FUNCTION_BLOCK MECHC_VIEWL (* Linear Mechanism View with Clamping & Local Data Publish/Subscribe *)
  (* Standard: 61499-1; Classification: View *)
  (* Version 0.2, 2004-10-06, JHC, Rockwell Automation, Added CNV input. *)
  (* Version 0.1, 2004-09-27, JHC, Rockwell Automation, Changed order of REND vars for consitency with MECH_VIEWL.. *)
  (* Version 0.0, 2002-05-21, JHC, Rockwell Automation, Copied/Modified from MECH_VIEWL. *)
  (* Compiler header: package fb.rt.mva; import fb.rt.net.*; *)
  (* Compiler classdef: public class MECHC_VIEWL extends FBMVCD *)
  (* Compiler Java Sun JDK 1.4.2 *)
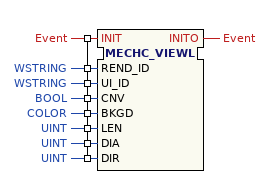
  EVENT_INPUT
    INIT WITH REND_ID, UI_ID, BKGD, LEN, DIA, DIR, CNV; (* Initialize *)
  END_EVENT
  EVENT_OUTPUT
    INITO; (* Initialized *)
  END_EVENT
  VAR_INPUT
    REND_ID : WSTRING; (* Rendering Data Channel from Model *)
    UI_ID : WSTRING; (* User Input Channel to Model *)
    CNV : BOOL; (* 0=Paint workpiece with clamp,1=Paint as conveyor with gate at end. *)
    BKGD : COLOR := blue; (* Background Color *)
    LEN : UINT; (* Length in Diameters *)
    DIA : UINT; (* Diameter *)
    DIR : UINT; (* Orientation:0=L/R,1=T/B,2=R/L,3=B/T *)
  END_VAR
  FBS
    REND : SUBL_4;
    VIEW : MECHC_VIEW;
    UI : PUBL_1;
  END_FBS
  EVENT_CONNECTIONS
    INIT TO REND.INIT;
    REND.INITO TO VIEW.INIT;
    VIEW.INITO TO UI.INIT;
    UI.INITO TO INITO;
    REND.IND TO VIEW.REQ;
    VIEW.IND TO UI.REQ;
  END_CONNECTIONS
  DATA_CONNECTIONS
    REND.RD_1 TO VIEW.POS;
    VIEW.FAULT TO UI.SD_1;
    REND_ID TO REND.ID;
    UI_ID TO UI.ID;
    BKGD TO VIEW.BKGD;
    LEN TO VIEW.LEN;
    DIA TO VIEW.DIA;
    DIR TO VIEW.DIR;
    REND.RD_2 TO VIEW.STYLE;
    REND.RD_3 TO VIEW.WKPC;
    REND.RD_4 TO VIEW.CLAMP;
    CNV TO VIEW.CNV;
  END_CONNECTIONS
END_FUNCTION_BLOCK
